TYPE T_Ctrl_SIf_GRN_Par :
STRUCT
END_STRUCT
END_TYPE

(* stored: Version 1.1.0.1, ProductVersion 3.1.0.25
   DUT T_Ctrl_SIf_GRN_Par: Id {acc58138-5a92-4dd5-a90e-bda48795aadd} *)
